// TIA Portal V20 export
DATA_BLOCK "BK03"   // DB192
// stored: MemoryReserve 100
   VAR
      "X10-1 ELECTRODE FIX LEFT TOP BACKWARD" : Bool;
      "X11-1 UNWINDER STOPPER BACKWARD" : Bool;
      "X12-1 ELECTRODE FIX LEFT BTM BACKWARD" : Bool;
      "X13-1 DIGITAL PRESSURE SWITCH OUT1" : Bool;
      "X14-1 ELECTRODE FIX LEFT TOP UP" : Bool;
      "X15-1 FRAME COVER BACKWARD" : Bool;
      "X16-1 ELECTRODE FIX LEFT BTM DOWN" : Bool;
      "X17-1 SPARE" : Bool;
      "X10-2 ELECTRODE FIX LEFT TOP FORWARD" : Bool;
      "X11-2 UNWINDER STOPPER FORWARD" : Bool;
      "X12-2 ELECTRODE FIX LEFT BTM FORWARD" : Bool;
      "X13-2 DIGITAL PRESSURE SWITCH OUT2" : Bool;
      "X14-2 ELECTRODE FIX LEFT TOP DOWN" : Bool;
      "X15-2 FRAME COVER FORWARD" : Bool;
      "X16-2 ELECTRODE FIX LEFT BTM UP" : Bool;
      "X17-2 SPARE" : Bool;
   END_VAR
BEGIN
END_DATA_BLOCK
